FUNCTION ifc_int : INT
VAR_INPUT
	Condition: BOOL;
	ValueTrue: INT;
	ValueFalse: INT;
END_VAR
VAR
END_VAR

IF Condition THEN
	ifc_int := ValueTrue;
ELSE
	ifc_int := ValueFalse;
END_IF

END_FUNCTION

(* stored: Version 1.1.0.1, ProductVersion 3.1.4024.6
   POU ifc_int: Id {4f1ae2a4-6bd4-4708-bce7-6aa733a65344}, SpecialFunc None *)
